TYPE TcoAbbRobotics_Status_v_1_x_x :
STRUCT
	ActionDescription : STRING(100);	
	State:TcoAbbRobotics_State_v_1_x_x;


END_STRUCT
END_TYPE

(* stored: Version 1.1.0.1, ProductVersion 3.1.4024.12
   DUT TcoAbbRobotics_Status_v_1_x_x: Id {f00768af-16ab-0d87-2aa7-e9ce54739eb7} *)
